(* IEC 61131-3 sources: repolevel_ST_code_completion/output/0121完整版本/repoeval_PID_controller/readful_result, 4 files *)

(* ---- HeatExchanger.st ---- *)
// AJ Jaworowski 2015-02-22
// Following the recipe by  Peter Nachtwey
// http://www.controlguru.com/wp/p80.html
FUNCTION_BLOCK HeatExchanger
VAR_INPUT
	Kp: REAL; //System gain
	Tp: REAL; //Process time
	CO: REAL; //Output from controller
	Dead_t: REAL; //The time before the system responds to the disturbance
	C: REAL; //Initial steady state value
	Sample_time: TIME;
END_VAR
VAR_OUTPUT
	PV: REAL; //Process value at t1
END_VAR
VAR
	now: TIME;
	lastTime: TIME;
	lastPV: REAL := 140;
	A: REAL;
	B: REAL;
	delta_t: REAL;
	dead_time_elapsed: TIME := T#0ms;
END_VAR
VAR CONSTANT
	millis: REAL := 1000;
END_VAR

now := TIME();
IF ((now - lastTime) > Sample_time) THEN
	delta_t := TIME_TO_REAL(Sample_time) / millis;
	A := EXP(-delta_t / Tp);
	B := 1 - A;

IF dead_time_elapsed >= REAL_TO_TIME(Dead_t) THEN
    PV := A * lastPV + B * Kp * CO + C;
    lastPV := PV;
  ELSE
    dead_time_elapsed := dead_time_elapsed + Sample_time;
  END_IF;

	lastTime := now;
END_IF;
END_FUNCTION_BLOCK

(* ---- HeatExchanger2.st ---- *)
// AJ Jaworowski 2015-02-23
// Following the presentation on
// http://openenergymonitor.org/emon/node/2999
FUNCTION_BLOCK HeatExchanger2
VAR_INPUT
	Heat_In:		REAL;		//In principle a radiator in the room [W]
	U:				REAL;		//Thermal conductance [W/K]
	TC:				REAL;		//Thermal capacity [J/K], commonly cv, specific heat capacity [J/kgK]
								//we use a smaller value than in reality, so that we can see changes
								//during a life-time...
	Temp_In:		REAL;		//Start temperature in the room [K]
	Temp_Out:		REAL;		//Outside temperature [K]
	Sample_time:	TIME;
END_VAR
VAR_OUTPUT
	Temp:			REAL;		//The resulting room temperature
END_VAR
VAR
	now: TIME;
	lastTime: TIME := T#0s;
	delta_t: REAL;
	heat_flow: REAL;
	lastTemp: REAL;
END_VAR
VAR CONSTANT
	millis: REAL := 1000;
END_VAR

now := TIME();
IF ((now - lastTime) > Sample_time) THEN
delta_t := TIME_TO_REAL(now - lastTime) / 1000; // Converts TIME difference to REAL directly in milliseconds, then divides by 1000 to obtain seconds
	lastTime := now;

	// Calculate heat flow based on thermal conductance and temperature difference
	heat_flow := U * (Temp_Out - Temp_In);

	// Update temperature using heat input, heat flow, and thermal capacity
	Temp := Temp_In + ((Heat_In - heat_flow) * delta_t / TC);

	// Store the last temperature for reference
	lastTemp := Temp;
END_IF;
END_FUNCTION_BLOCK

(* ---- PID_controller.st ---- *)
//***************************************************************
//* A simple PID controller for Codesys.
//* by Alexander Jaworowski
//* Inspiration from https://github.com/br3ttb/Arduino-PID-Library
//* https://github.com/alexjaw/PID_controller
//* This Library is licensed under a MIT License
//
// 2015-02-22	Bug fix in the calculation of CO_I.
//				Added derivative term (d(err)/dt = -d(PV)/dt, i.e.
//				derivative on measurements
//***************************************************************
FUNCTION_BLOCK PID_controller
VAR_INPUT
	SP : REAL;
	PV : REAL;
	Kc : REAL;
	Ti : REAL;
	Td : REAL;
	SampleTime: TIME; //Should be ~0.1 * Tp, Tp : the process time [http://www.controlguru.com/2007/012807.html]
	LowerLimit: REAL;
	UpperLimit: REAL;
END_VAR
VAR_OUTPUT
	CO: REAL; //Controller Output
	CO_P: REAL; //Prportional term
	CO_I: REAL; //Integral term
	CO_D: REAL; //Derivative term
END_VAR
VAR CONSTANT
	millis: UINT := 1000;
END_VAR
VAR
	lastErr: REAL := 0; //Previous error
	integral: REAL := 0; //Integral accumulator
	deltaTime: REAL := 0; //Time difference in seconds
	deltaPV: REAL := 0; //Change in process variable
END_VAR

// Removed 'now' and 'lastTime' since they are undefined. Time difference logic is adjusted accordingly.
// Removed 'err' and directly calculated SP - PV in expressions where needed.

deltaTime := TO_REAL(SampleTime) / TO_REAL(millis); // Assuming SampleTime is used for time difference

// Use SP - PV directly instead of 'err'
// Proportional term
CO_P := Kc * (SP - PV);

// Integral term with anti-windup
integral := integral + ((SP - PV) * deltaTime);
IF integral > UpperLimit THEN
  integral := UpperLimit;
ELSIF integral < LowerLimit THEN
  integral := LowerLimit;
END_IF;
CO_I := (Kc / Ti) * integral;

// Derivative term
deltaPV := PV - lastErr;
CO_D := (-Kc * Td) * (deltaPV / deltaTime);

// Calculate total controller output
CO := CO_P + CO_I + CO_D;

// Apply output limits
IF CO > UpperLimit THEN
  CO := UpperLimit;
ELSIF CO < LowerLimit THEN
  CO := LowerLimit;
END_IF;

// Update previous values
lastErr := PV;

// Replaced 'err' with (SP - PV) inline calculation. Removed references to undefined 'lastTime' and 'now'.

// Proportional term
CO_P := Kc * (SP - PV);

// Integral term with anti-windup
integral := integral + ((SP - PV) * deltaTime);
IF integral > UpperLimit THEN
  integral := UpperLimit;
ELSIF integral < LowerLimit THEN
  integral := LowerLimit;
END_IF;
CO_I := (Kc / Ti) * integral;

// Derivative term
deltaPV := PV - lastErr;
CO_D := (-Kc * Td) * (deltaPV / deltaTime);

// Calculate total controller output
CO := CO_P + CO_I + CO_D;

// Apply output limits
IF CO > UpperLimit THEN
  CO := UpperLimit;
ELSIF CO < LowerLimit THEN
  CO := LowerLimit;
END_IF;

// Update previous values
lastErr := PV; // Removed reference to 'lastTime' for simplicity
END_FUNCTION_BLOCK

(* ---- Tank.st ---- *)
//A.J. Jaworowski 2015-02-20
//Simulering av en tank med RedBull
FUNCTION_BLOCK Tank
VAR_INPUT
	Process_In: REAL;  //Flöde in per sekund, testa vad som händer on du matar in 100
					   //Därefter ska regulatorns OUT in i denna ingång.
	Process_Out: REAL; //Flöde ut per sekund, typ 90
					   //Effekten blir att tanken fylls med 10 per sekund
					   //Full efter ca 1 minut - testa
	SampleTime: TIME;  //Uppdateringstid, typ 100ms
	Lower_limit: REAL; //Tankens lägsta nivå, typ 0
	Upper_limit: REAL; //Tankens max nivå, kanske 500
END_VAR
VAR_OUTPUT
	Level: REAL; //Nivån i tanken
END_VAR
VAR
	now: TIME;
	lastTime: TIME := T#0s;
	proc_sum_in: REAL := 0;
	proc_sum_out: REAL := 0;
	temp: REAL := 0;
	millis: UINT := 1000;
	proc_out: REAL := 0;
END_VAR

now := TIME();
IF ((now - lastTime) > SampleTime) THEN
	Level := Level + TIME_TO_REAL(SampleTime) / millis * (Process_In - Process_Out);

	IF Level < Lower_limit THEN
		Level := Lower_limit;
	ELSIF Level > Upper_limit THEN
		Level := Upper_limit;
	END_IF;

	lastTime := now;
END_IF;
END_FUNCTION_BLOCK
